Yaskawa INFORM job: R1_W12(125,90)(KAMERA).JBI

/JOB
//NAME R1_W12(125,90)(KAMERA)
//POS
///NPOS 15,15,0,0,0,0
///TOOL 0
///POSTYPE PULSE
///PULSE
C00000=-167342,-92471,-131631,15300,65044,71165
C00001=-162457,-153227,-130225,-463,96631,68116
C00002=-17388,-168806,-111585,-4698,65840,-53499
C00003=56151,-123607,-84681,-24015,93824,-29050
C00004=38514,-119451,-74638,-22450,88065,-28099
C00005=47917,-112097,-69645,-23905,91780,-24333
C00006=-60796,-15342,30656,25990,89314,17670
C00007=-59751,-12665,34197,26363,88297,17792
C00008=34505,-120946,-73457,-26839,85825,-27870
C00009=16114,-121307,-68615,-34025,78747,-32161
C00010=16104,-135523,-87595,-33683,82412,-33282
C00011=16104,-134772,-86650,-33694,82248,-33232
C00012=16104,-134772,-86650,-33694,82248,81437
C00013=16104,-134772,-86650,-33694,-810,81437
C00014=17357,-183139,-134392,-16915,3390,73963
BC00000=335588,15,1060137
BC00001=316378,15,1014256
BC00002=207039,196,620236
BC00003=205412,4,249661
BC00004=159623,24,288253
BC00005=154111,4,249661
BC00006=113659,15,530075
BC00007=113659,15,530075
BC00008=154111,4,249661
BC00009=154111,4,249661
BC00010=154111,4,249661
BC00011=154111,4,768006
BC00012=154111,4,768006
BC00013=154111,4,768006
BC00014=154111,3790,1028555
//INST
///DATE 2024/11/28 10:08
///ATTR SC,RW
///GROUP1 RB1,BS1
NOP
'r1_W12(125,90)(kamera)
'Path W411
SFTOF
MOVJ C00000 BC00000 VJ=100.00
MOVJ C00001 BC00001 VJ=100.00
MOVJ C00002 BC00002 VJ=100.00
MOVJ C00003 BC00003 VJ=100.00
MOVJ C00004 BC00004 VJ=100.00
MOVJ C00005 BC00005 VJ=15.00 PL=0
REFP 1 C00006 BC00006
REFP 2 C00007 BC00007
MACRO1 MJ#(0) ARGF6
ARCON
WVON WEV#(14)
MOVL C00008 BC00008 V=10.8
MOVL C00009 BC00009 V=10.8
ARCOF
WVOF
MOVL C00010 BC00010 V=100.0
MOVL C00011 BC00011 V=333.3
MOVJ C00012 BC00012 VJ=100.00
MOVJ C00013 BC00013 VJ=100.00
MOVJ C00014 BC00014 VJ=100.00
'Path W412
SFTOF
'W27-1
END
